ABB RAPID module: traj1smoothed.MOD

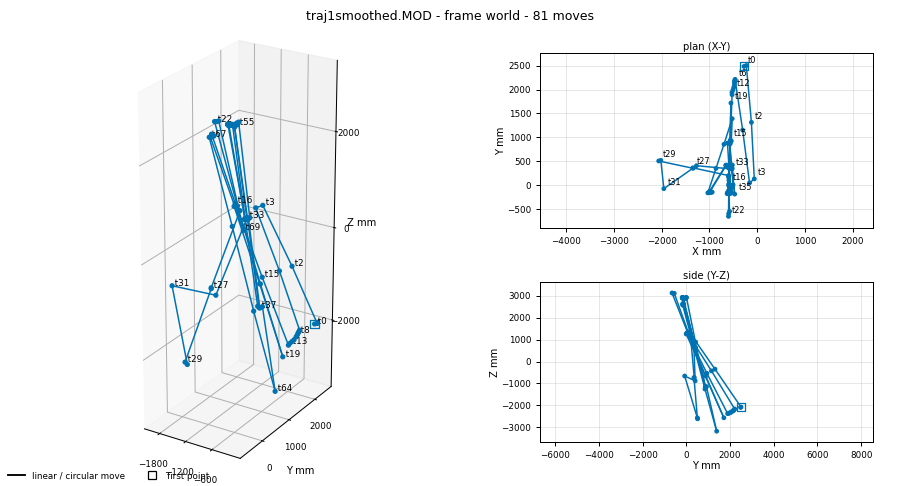
[picture p0: tool path of traj1smoothed.MOD in frame world, 81 of 82 moves have a stored position in this frame; points joined in program order, loops and branches not executed]
MODULE MainModule
PERS tooldata Servo:=[TRUE,[[0,0,114.2],[1,0,0,0]],[0.215,[8.7,12.3,49.2],[1,0,0,0],0.00021,0.00024,0.00009]];
PERS tooldata tObject:=[TRUE,[[0,0,130],[0.707106781,-0.707106781,0,0]],[0.215,[8.7,12.3,49.2],[1,0,0,0],0.00021,0.00024,0.00009]];
PERS wobjdata handpos:= [FALSE,TRUE,"",[[-400,0,250],[1,0,0,0]],[[0,0,0],[1,0,0,0]]];
    PROC main()
        ConfL\Off;
        SingArea\Wrist;
        !Startpos
        MoveAbsJ [[0.441359,-16.418,10.8814,2.79121,60.2034,-14.3875],[168.362,9E+09,9E+09,9E+09,9E+09,9E+09]] \NoEOffs, v1000, fine, wi_tGripper;
        path;
    ENDPROC
    PROC path()

VAR robtarget t0 := [[123.45197327880837, 2483.780227785589, -2348.344137061463], [0, -1, 0, 0], [0,0,-1,4], [-96,9E+09,9E+09,9E+09,9E+09,9E+09]];
VAR robtarget t1 := [[172.0670230010615, 2502.808697034114, -2332.24679612455], [0, -1, 0, 0], [0,0,-1,4], [-96,9E+09,9E+09,9E+09,9E+09,9E+09]];
VAR robtarget t2 := [[278.2773550958402, 1313.750269544781, -598.3539635779312], [0, -1, 0, 0], [0,0,-1,4], [-96,9E+09,9E+09,9E+09,9E+09,9E+09]];
VAR robtarget t3 := [[338.90898794341996, 130.62076047011854, 1102.0424095735846], [0, -1, 0, 0], [0,0,-1,4], [-96,9E+09,9E+09,9E+09,9E+09,9E+09]];
VAR robtarget t4 := [[239.31131677510967, 46.01081850908662, 1059.8490608023326], [0, -1, 0, 0], [0,0,-1,4], [-96,9E+09,9E+09,9E+09,9E+09,9E+09]];
VAR robtarget t5 := [[95.30462700221017, 1152.38697204331, -678.8853084480063], [0, -1, 0, 0], [0,0,-1,4], [-96,9E+09,9E+09,9E+09,9E+09,9E+09]];
VAR robtarget t6 := [[-63.36910785979792, 2213.9973893918595, -2420.5022973796886], [0, -1, 0, 0], [0,0,-1,4], [-96,9E+09,9E+09,9E+09,9E+09,9E+09]];
VAR robtarget t7 := [[-65.17321560227712, 2191.048596103816, -2448.2274115828395], [0, -1, 0, 0], [0,0,-1,4], [-96,9E+09,9E+09,9E+09,9E+09,9E+09]];
VAR robtarget t8 := [[-71.56162519990338, 2175.2346300780814, -2468.193989987165], [0, -1, 0, 0], [0,0,-1,4], [-96,9E+09,9E+09,9E+09,9E+09,9E+09]];
VAR robtarget t9 := [[-76.9983175239739, 2155.607321650718, -2499.71661387214], [0, -1, 0, 0], [0,0,-1,4], [-96,9E+09,9E+09,9E+09,9E+09,9E+09]];
VAR robtarget t10 := [[-76.31520794936695, 2103.645900585614, -2526.7961936744273], [0, -1, 0, 0], [0,0,-1,4], [-96,9E+09,9E+09,9E+09,9E+09,9E+09]];
VAR robtarget t11 := [[-91.26198794302982, 2047.3288034263858, -2573.389881322257], [0, -1, 0, 0], [0,0,-1,4], [-96,9E+09,9E+09,9E+09,9E+09,9E+09]];
VAR robtarget t12 := [[-107.3130126249458, 1991.352495111901, -2594.6104473912847], [0, -1, 0, 0], [0,0,-1,4], [-96,9E+09,9E+09,9E+09,9E+09,9E+09]];
VAR robtarget t13 := [[-128.96132520964585, 1939.0077314152172, -2621.1257880884805], [0, -1, 0, 0], [0,0,-1,4], [-96,9E+09,9E+09,9E+09,9E+09,9E+09]];
VAR robtarget t14 := [[-125.6757865163689, 1891.7416972133587, -2633.421109839484], [0, -1, 0, 0], [0,0,-1,4], [-96,9E+09,9E+09,9E+09,9E+09,9E+09]];
VAR robtarget t15 := [[-162.31089879533124, 943.5157765321271, -792.0949508080666], [0, -1, 0, 0], [0,0,-1,4], [-96,9E+09,9E+09,9E+09,9E+09,9E+09]];
VAR robtarget t16 := [[-193.89590738735384, 25.726263998332, 1058.834661495532], [0, -1, 0, 0], [0,0,-1,4], [-96,9E+09,9E+09,9E+09,9E+09,9E+09]];
VAR robtarget t17 := [[-198.62085110692982, -4.477175700340341, 1009.1428394800721], [0, -1, 0, 0], [0,0,-1,4], [-96,9E+09,9E+09,9E+09,9E+09,9E+09]];
VAR robtarget t18 := [[-169.6531598146668, 865.1205052705678, -901.9879179559268], [0, -1, 0, 0], [0,0,-1,4], [-96,9E+09,9E+09,9E+09,9E+09,9E+09]];
VAR robtarget t19 := [[-149.6958240431798, 1717.930633624114, -2823.3620024852316], [0, -1, 0, 0], [0,0,-1,4], [-96,9E+09,9E+09,9E+09,9E+09,9E+09]];
VAR robtarget t20 := [[-169.6756018707418, 888.4425795232621, -914.5769749366513], [0, -1, 0, 0], [0,0,-1,4], [-96,9E+09,9E+09,9E+09,9E+09,9E+09]];
VAR robtarget t21 := [[-192.15914337238237, 101.21945473498606, 979.3423329932617], [0, -1, 0, 0], [0,0,-1,4], [-96,9E+09,9E+09,9E+09,9E+09,9E+09]];
VAR robtarget t22 := [[-201.1830156164082, -653.5722365528959, 2887.851725420608], [0, -1, 0, 0], [0,0,-1,4], [-96,9E+09,9E+09,9E+09,9E+09,9E+09]];
VAR robtarget t23 := [[-196.98146133427508, -596.0507051176519, 2868.520572012061], [0, -1, 0, 0], [0,0,-1,4], [-96,9E+09,9E+09,9E+09,9E+09,9E+09]];
VAR robtarget t24 := [[-179.0254582118774, -550.4853804920127, 2869.110064489453], [0, -1, 0, 0], [0,0,-1,4], [-96,9E+09,9E+09,9E+09,9E+09,9E+09]];
VAR robtarget t25 := [[-199.87164277033122, 168.80811452867698, 863.3402049612712], [0, -1, 0, 0], [0,0,-1,4], [-96,9E+09,9E+09,9E+09,9E+09,9E+09]];
VAR robtarget t26 := [[-199.83948017692023, 200.53421548431308, 846.5530305744547], [0, -1, 0, 0], [0,0,-1,4], [-96,9E+09,9E+09,9E+09,9E+09,9E+09]];
VAR robtarget t27 := [[-947.5598868965106, 361.9296308424034, -978.4613651276785], [0, -1, 0, 0], [0,0,-1,4], [-96,9E+09,9E+09,9E+09,9E+09,9E+09]];
VAR robtarget t28 := [[-941.7151957916036, 352.2407347860694, -992.6785638373589], [0, -1, 0, 0], [0,0,-1,4], [-96,9E+09,9E+09,9E+09,9E+09,9E+09]];
VAR robtarget t29 := [[-1661.5282499685884, 505.16917363828594, -2824.7509483979], [0, -1, 0, 0], [0,0,-1,4], [-96,9E+09,9E+09,9E+09,9E+09,9E+09]];
VAR robtarget t30 := [[-1617.0080528765757, 517.5373022143422, -2870.04617187687], [0, -1, 0, 0], [0,0,-1,4], [-96,9E+09,9E+09,9E+09,9E+09,9E+09]];
VAR robtarget t31 := [[-1553.9069316208634, -73.79109378893207, -913.5993323327], [0, -1, 0, 0], [0,0,-1,4], [-96,9E+09,9E+09,9E+09,9E+09,9E+09]];
VAR robtarget t32 := [[-870.7794370177955, 406.5667497109633, -1134.7561205239003], [0, -1, 0, 0], [0,0,-1,4], [-96,9E+09,9E+09,9E+09,9E+09,9E+09]];
VAR robtarget t33 := [[-129.7359237290919, 337.3424201451147, 665.6093470046382], [0, -1, 0, 0], [0,0,-1,4], [-96,9E+09,9E+09,9E+09,9E+09,9E+09]];
VAR robtarget t34 := [[-142.6333367822861, 350.7778576213944, 659.6542290808931], [0, -1, 0, 0], [0,0,-1,4], [-96,9E+09,9E+09,9E+09,9E+09,9E+09]];
VAR robtarget t35 := [[-71.09616720793116, -187.751839665803, 2656.3167897829635], [0, -1, 0, 0], [0,0,-1,4], [-96,9E+09,9E+09,9E+09,9E+09,9E+09]];
VAR robtarget t36 := [[-124.18371818133171, 353.1588170244417, 623.4753396663407], [0, -1, 0, 0], [0,0,-1,4], [-96,9E+09,9E+09,9E+09,9E+09,9E+09]];
VAR robtarget t37 := [[-185.253150469207, 873.9992695082627, -1412.1085010282707], [0, -1, 0, 0], [0,0,-1,4], [-96,9E+09,9E+09,9E+09,9E+09,9E+09]];
VAR robtarget t38 := [[-222.4853859890584, 880.6988326998469, -1396.0004353729908], [0, -1, 0, 0], [0,0,-1,4], [-96,9E+09,9E+09,9E+09,9E+09,9E+09]];
VAR robtarget t39 := [[-189.6298267133733, 363.0193546707583, 636.2791703178914], [0, -1, 0, 0], [0,0,-1,4], [-96,9E+09,9E+09,9E+09,9E+09,9E+09]];
VAR robtarget t40 := [[-141.96919537845292, -147.91308173457537, 2683.575571924676], [0, -1, 0, 0], [0,0,-1,4], [-96,9E+09,9E+09,9E+09,9E+09,9E+09]];
VAR robtarget t41 := [[-144.2807050432762, -164.63165505603342, 2674.93970895107], [0, -1, 0, 0], [0,0,-1,4], [-96,9E+09,9E+09,9E+09,9E+09,9E+09]];
VAR robtarget t42 := [[-169.63554081179575, -177.67226905725764, 2677.542151250687], [0, -1, 0, 0], [0,0,-1,4], [-96,9E+09,9E+09,9E+09,9E+09,9E+09]];
VAR robtarget t43 := [[-195.3508934236626, -180.5134840605642, 2672.1635994198514], [0, -1, 0, 0], [0,0,-1,4], [-96,9E+09,9E+09,9E+09,9E+09,9E+09]];
VAR robtarget t44 := [[-209.09830808143357, -173.2064662482046, 2679.8461386164286], [0, -1, 0, 0], [0,0,-1,4], [-96,9E+09,9E+09,9E+09,9E+09,9E+09]];
VAR robtarget t45 := [[-227.3581923429079, -179.4710413959663, 2679.0978130301987], [0, -1, 0, 0], [0,0,-1,4], [-96,9E+09,9E+09,9E+09,9E+09,9E+09]];
VAR robtarget t46 := [[-228.5514670205092, -173.09828721280152, 2673.361172173061], [0, -1, 0, 0], [0,0,-1,4], [-96,9E+09,9E+09,9E+09,9E+09,9E+09]];
VAR robtarget t47 := [[-222.97576289509837, -168.87070480134724, 2657.8597637829985], [0, -1, 0, 0], [0,0,-1,4], [-96,9E+09,9E+09,9E+09,9E+09,9E+09]];
VAR robtarget t48 := [[-187.40448600537542, 359.59636265319705, 623.7528732021439], [0, -1, 0, 0], [0,0,-1,4], [-96,9E+09,9E+09,9E+09,9E+09,9E+09]];
VAR robtarget t49 := [[-189.91977282775926, 350.6535409547082, 620.6313028595152], [0, -1, 0, 0], [0,0,-1,4], [-96,9E+09,9E+09,9E+09,9E+09,9E+09]];
VAR robtarget t50 := [[-183.19398350324013, 355.67364703901404, 619.2996040284754], [0, -1, 0, 0], [0,0,-1,4], [-96,9E+09,9E+09,9E+09,9E+09,9E+09]];
VAR robtarget t51 := [[-210.0320304278792, -157.83324578597555, 2644.3505127391627], [0, -1, 0, 0], [0,0,-1,4], [-96,9E+09,9E+09,9E+09,9E+09,9E+09]];
VAR robtarget t52 := [[-213.46183196310977, -144.05743890136876, 2642.4967231260175], [0, -1, 0, 0], [0,0,-1,4], [-96,9E+09,9E+09,9E+09,9E+09,9E+09]];
VAR robtarget t53 := [[-195.03038705015618, -110.98127875062085, 2641.6439287699473], [0, -1, 0, 0], [0,0,-1,4], [-96,9E+09,9E+09,9E+09,9E+09,9E+09]];
VAR robtarget t54 := [[-152.59778212721966, -72.95478043908155, 2637.198912088225], [0, -1, 0, 0], [0,0,-1,4], [-96,9E+09,9E+09,9E+09,9E+09,9E+09]];
VAR robtarget t55 := [[-113.0359564899629, -26.566690992573434, 2640.7971971548805], [0, -1, 0, 0], [0,0,-1,4], [-96,9E+09,9E+09,9E+09,9E+09,9E+09]];
VAR robtarget t56 := [[-121.67024429090301, -14.997889546826052, 2649.3462199597125], [0, -1, 0, 0], [0,0,-1,4], [-96,9E+09,9E+09,9E+09,9E+09,9E+09]];
VAR robtarget t57 := [[-137.48278172829905, -18.260542559761433, 2654.3748469656357], [0, -1, 0, 0], [0,0,-1,4], [-96,9E+09,9E+09,9E+09,9E+09,9E+09]];
VAR robtarget t58 := [[-133.6672849697944, -14.204175910826196, 2666.910880672061], [0, -1, 0, 0], [0,0,-1,4], [-96,9E+09,9E+09,9E+09,9E+09,9E+09]];
VAR robtarget t59 := [[-106.13439677313141, 6.920296362909546, 2684.785104595534], [0, -1, 0, 0], [0,0,-1,4], [-96,9E+09,9E+09,9E+09,9E+09,9E+09]];
VAR robtarget t60 := [[-120.22564348824234, 419.7268598686734, 642.2478530800479], [0, -1, 0, 0], [0,0,-1,4], [-96,9E+09,9E+09,9E+09,9E+09,9E+09]];
VAR robtarget t61 := [[-146.76090985604395, 412.38629942703886, 637.636695455018], [0, -1, 0, 0], [0,0,-1,4], [-96,9E+09,9E+09,9E+09,9E+09,9E+09]];
VAR robtarget t62 := [[-168.22219514450828, 869.6795051912934, -1417.263274998179], [0, -1, 0, 0], [0,0,-1,4], [-96,9E+09,9E+09,9E+09,9E+09,9E+09]];
VAR robtarget t63 := [[-142.71273678580334, 923.7733665828956, -1401.5053807477334], [0, -1, 0, 0], [0,0,-1,4], [-96,9E+09,9E+09,9E+09,9E+09,9E+09]];
VAR robtarget t64 := [[-123.22935419906366, 1390.0893522125646, -3438.114403516943], [0, -1, 0, 0], [0,0,-1,4], [-96,9E+09,9E+09,9E+09,9E+09,9E+09]];
VAR robtarget t65 := [[-296.15846836957445, 854.5565732043196, -1508.6317753216533], [0, -1, 0, 0], [0,0,-1,4], [-96,9E+09,9E+09,9E+09,9E+09,9E+09]];
VAR robtarget t66 := [[-463.0243786654314, 349.66460443276065, 414.7391125086879], [0, -1, 0, 0], [0,0,-1,4], [-96,9E+09,9E+09,9E+09,9E+09,9E+09]];
VAR robtarget t67 := [[-633.4674899693175, -162.24505635139838, 2337.5562191339122], [0, -1, 0, 0], [0,0,-1,4], [-96,9E+09,9E+09,9E+09,9E+09,9E+09]];
VAR robtarget t68 := [[-611.942871282688, -150.69536035716865, 2327.486775599343], [0, -1, 0, 0], [0,0,-1,4], [-96,9E+09,9E+09,9E+09,9E+09,9E+09]];
VAR robtarget t69 := [[-258.6611317221678, 412.904242714683, 358.13155201903896], [0, -1, 0, 0], [0,0,-1,4], [-96,9E+09,9E+09,9E+09,9E+09,9E+09]];
VAR robtarget t70 := [[-251.75807989991816, 414.7654563521526, 371.9114588417323], [0, -1, 0, 0], [0,0,-1,4], [-96,9E+09,9E+09,9E+09,9E+09,9E+09]];
VAR robtarget t71 := [[-246.74145905228775, 419.6815736393265, 385.3638037425684], [0, -1, 0, 0], [0,0,-1,4], [-96,9E+09,9E+09,9E+09,9E+09,9E+09]];
VAR robtarget t72 := [[-586.9071702734813, -134.34844408419278, 2364.899585025393], [0, -1, 0, 0], [0,0,-1,4], [-96,9E+09,9E+09,9E+09,9E+09,9E+09]];
VAR robtarget t73 := [[-579.8306670631828, -131.90380045754833, 2360.3086468033093], [0, -1, 0, 0], [0,0,-1,4], [-96,9E+09,9E+09,9E+09,9E+09,9E+09]];
VAR robtarget t74 := [[-582.6633868022558, -127.281470022346, 2365.0437853634007], [0, -1, 0, 0], [0,0,-1,4], [-96,9E+09,9E+09,9E+09,9E+09,9E+09]];
VAR robtarget t75 := [[-592.61255465612, -137.74245984041963, 2374.2804220456205], [0, -1, 0, 0], [0,0,-1,4], [-96,9E+09,9E+09,9E+09,9E+09,9E+09]];
VAR robtarget t76 := [[-587.5732602333875, -142.42272299906165, 2387.2543915871543], [0, -1, 0, 0], [0,0,-1,4], [-96,9E+09,9E+09,9E+09,9E+09,9E+09]];
VAR robtarget t77 := [[-590.1349932352252, -151.32509094208802, 2403.2844413028315], [0, -1, 0, 0], [0,0,-1,4], [-96,9E+09,9E+09,9E+09,9E+09,9E+09]];
VAR robtarget t78 := [[-573.8296063618772, -151.25169531888085, 2388.5156493513437], [0, -1, 0, 0], [0,0,-1,4], [-96,9E+09,9E+09,9E+09,9E+09,9E+09]];
VAR robtarget t79 := [[-561.1495065573185, -149.51684121345644, 2378.2977019121263], [0, -1, 0, 0], [0,0,-1,4], [-96,9E+09,9E+09,9E+09,9E+09,9E+09]];
VAR robtarget t80 := [[-542.4912901793865, -146.14921466275973, 2374.4911832227767], [0, -1, 0, 0], [0,0,-1,4], [-96,9E+09,9E+09,9E+09,9E+09,9E+09]];MoveL t0, v100\V:=100.000, z1, wi_tGripper, \WObj:=handpos;
MoveL t1, v100\V:=100.000, z1, wi_tGripper, \WObj:=handpos;
MoveL t2, v100\V:=100.000, z1, wi_tGripper, \WObj:=handpos;
MoveL t3, v100\V:=100.000, z1, wi_tGripper, \WObj:=handpos;
MoveL t4, v100\V:=100.000, z1, wi_tGripper, \WObj:=handpos;
MoveL t5, v100\V:=100.000, z1, wi_tGripper, \WObj:=handpos;
MoveL t6, v100\V:=100.000, z1, wi_tGripper, \WObj:=handpos;
MoveL t7, v100\V:=100.000, z1, wi_tGripper, \WObj:=handpos;
MoveL t8, v100\V:=100.000, z1, wi_tGripper, \WObj:=handpos;
MoveL t9, v100\V:=100.000, z1, wi_tGripper, \WObj:=handpos;
MoveL t10, v100\V:=100.000, z1, wi_tGripper, \WObj:=handpos;
MoveL t11, v100\V:=100.000, z1, wi_tGripper, \WObj:=handpos;
MoveL t12, v100\V:=100.000, z1, wi_tGripper, \WObj:=handpos;
MoveL t13, v100\V:=100.000, z1, wi_tGripper, \WObj:=handpos;
MoveL t14, v100\V:=100.000, z1, wi_tGripper, \WObj:=handpos;
MoveL t15, v100\V:=100.000, z1, wi_tGripper, \WObj:=handpos;
MoveL t16, v100\V:=100.000, z1, wi_tGripper, \WObj:=handpos;
MoveL t17, v100\V:=100.000, z1, wi_tGripper, \WObj:=handpos;
MoveL t18, v100\V:=100.000, z1, wi_tGripper, \WObj:=handpos;
MoveL t19, v100\V:=100.000, z1, wi_tGripper, \WObj:=handpos;
MoveL t20, v100\V:=100.000, z1, wi_tGripper, \WObj:=handpos;
MoveL t21, v100\V:=100.000, z1, wi_tGripper, \WObj:=handpos;
MoveL t22, v100\V:=100.000, z1, wi_tGripper, \WObj:=handpos;
MoveL t23, v100\V:=100.000, z1, wi_tGripper, \WObj:=handpos;
MoveL t24, v100\V:=100.000, z1, wi_tGripper, \WObj:=handpos;
MoveL t25, v100\V:=100.000, z1, wi_tGripper, \WObj:=handpos;
MoveL t26, v100\V:=100.000, z1, wi_tGripper, \WObj:=handpos;
MoveL t27, v100\V:=100.000, z1, wi_tGripper, \WObj:=handpos;
MoveL t28, v100\V:=100.000, z1, wi_tGripper, \WObj:=handpos;
MoveL t29, v100\V:=100.000, z1, wi_tGripper, \WObj:=handpos;
MoveL t30, v100\V:=100.000, z1, wi_tGripper, \WObj:=handpos;
MoveL t31, v100\V:=100.000, z1, wi_tGripper, \WObj:=handpos;
MoveL t32, v100\V:=100.000, z1, wi_tGripper, \WObj:=handpos;
MoveL t33, v100\V:=100.000, z1, wi_tGripper, \WObj:=handpos;
MoveL t34, v100\V:=100.000, z1, wi_tGripper, \WObj:=handpos;
MoveL t35, v100\V:=100.000, z1, wi_tGripper, \WObj:=handpos;
MoveL t36, v100\V:=100.000, z1, wi_tGripper, \WObj:=handpos;
MoveL t37, v100\V:=100.000, z1, wi_tGripper, \WObj:=handpos;
MoveL t38, v100\V:=100.000, z1, wi_tGripper, \WObj:=handpos;
MoveL t39, v100\V:=100.000, z1, wi_tGripper, \WObj:=handpos;
MoveL t40, v100\V:=100.000, z1, wi_tGripper, \WObj:=handpos;
MoveL t41, v100\V:=100.000, z1, wi_tGripper, \WObj:=handpos;
MoveL t42, v100\V:=100.000, z1, wi_tGripper, \WObj:=handpos;
MoveL t43, v100\V:=100.000, z1, wi_tGripper, \WObj:=handpos;
MoveL t44, v100\V:=100.000, z1, wi_tGripper, \WObj:=handpos;
MoveL t45, v100\V:=100.000, z1, wi_tGripper, \WObj:=handpos;
MoveL t46, v100\V:=100.000, z1, wi_tGripper, \WObj:=handpos;
MoveL t47, v100\V:=100.000, z1, wi_tGripper, \WObj:=handpos;
MoveL t48, v100\V:=100.000, z1, wi_tGripper, \WObj:=handpos;
MoveL t49, v100\V:=100.000, z1, wi_tGripper, \WObj:=handpos;
MoveL t50, v100\V:=100.000, z1, wi_tGripper, \WObj:=handpos;
MoveL t51, v100\V:=100.000, z1, wi_tGripper, \WObj:=handpos;
MoveL t52, v100\V:=100.000, z1, wi_tGripper, \WObj:=handpos;
MoveL t53, v100\V:=100.000, z1, wi_tGripper, \WObj:=handpos;
MoveL t54, v100\V:=100.000, z1, wi_tGripper, \WObj:=handpos;
MoveL t55, v100\V:=100.000, z1, wi_tGripper, \WObj:=handpos;
MoveL t56, v100\V:=100.000, z1, wi_tGripper, \WObj:=handpos;
MoveL t57, v100\V:=100.000, z1, wi_tGripper, \WObj:=handpos;
MoveL t58, v100\V:=100.000, z1, wi_tGripper, \WObj:=handpos;
MoveL t59, v100\V:=100.000, z1, wi_tGripper, \WObj:=handpos;
MoveL t60, v100\V:=100.000, z1, wi_tGripper, \WObj:=handpos;
MoveL t61, v100\V:=100.000, z1, wi_tGripper, \WObj:=handpos;
MoveL t62, v100\V:=100.000, z1, wi_tGripper, \WObj:=handpos;
MoveL t63, v100\V:=100.000, z1, wi_tGripper, \WObj:=handpos;
MoveL t64, v100\V:=100.000, z1, wi_tGripper, \WObj:=handpos;
MoveL t65, v100\V:=100.000, z1, wi_tGripper, \WObj:=handpos;
MoveL t66, v100\V:=100.000, z1, wi_tGripper, \WObj:=handpos;
MoveL t67, v100\V:=100.000, z1, wi_tGripper, \WObj:=handpos;
MoveL t68, v100\V:=100.000, z1, wi_tGripper, \WObj:=handpos;
MoveL t69, v100\V:=100.000, z1, wi_tGripper, \WObj:=handpos;
MoveL t70, v100\V:=100.000, z1, wi_tGripper, \WObj:=handpos;
MoveL t71, v100\V:=100.000, z1, wi_tGripper, \WObj:=handpos;
MoveL t72, v100\V:=100.000, z1, wi_tGripper, \WObj:=handpos;
MoveL t73, v100\V:=100.000, z1, wi_tGripper, \WObj:=handpos;
MoveL t74, v100\V:=100.000, z1, wi_tGripper, \WObj:=handpos;
MoveL t75, v100\V:=100.000, z1, wi_tGripper, \WObj:=handpos;
MoveL t76, v100\V:=100.000, z1, wi_tGripper, \WObj:=handpos;
MoveL t77, v100\V:=100.000, z1, wi_tGripper, \WObj:=handpos;
MoveL t78, v100\V:=100.000, z1, wi_tGripper, \WObj:=handpos;
MoveL t79, v100\V:=100.000, z1, wi_tGripper, \WObj:=handpos;
MoveL t80, v100\V:=100.000, z1, wi_tGripper, \WObj:=handpos;

ENDPROC
ENDMODULE
